TYPE structHMIGlobal :
STRUCT
	hmi:structHMI;
	btns:structHMIBtns;
	GlobalMessages:structHMIMessages;
	
END_STRUCT
END_TYPE

(* stored: Version 1.1.0.1, ProductVersion 3.1.4024.11
   DUT structHMIGlobal: Id {37d41432-a392-0549-053b-072300f99ec8} *)
